// SIMATIC S7-200 project (STEP 7-Micro/WIN), CPU 221 REL 01.10

SYMBOL_TABLE USR1
Always_On        SM0.0    // This bit is always on.
Final_Count      VW0      // Variable memory word VW0 contains the ending value in the loop count (FINAL).
Initial_Count    VW10     // Variable memory word VW10 contains starting value in the loop count (INITIAL).
Current_Count    VW20     // Variable memory word VW20 contains the current loop count (INDEX).
First_Address    VB100    // Variable memory byte VB100 is the first address under which a value is saved.
END_SYMBOL_TABLE

ORGANIZATION_BLOCK MAIN:OB1
TITLE=
//  题目：设置位或字节的几种方法
// ***概述***
// 本程序描述了用一定值存入预定的存储区域或对预定的存储区域清零的几种方法
// 采用下列指令：
// *FILL           指令
// *FOR...NEXT     循环指令
// *RESET          指令
// 
// ***程序和注释***
// 本程序描述了用一定值存入预定的存储器位或字节，以及清除存储区内容的几种方法
// 采用下列指令：
// FILL          设置一个或几个字
// FOR...NEXT    FOR...NEXT循环
// R             对一位或几位置 0
// 
BEGIN
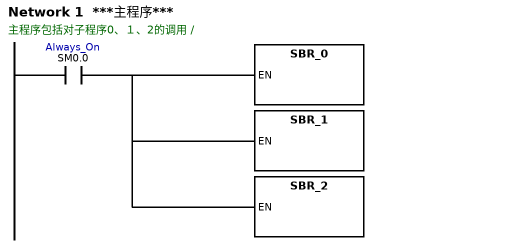
Network 1 // ***主程序***
// 主程序包括对子程序0、１、2的调用
// 
// SM0.0总是1
// 调用子程序0（FILL）
// 调用子程序1.（FOR...NEXT）
// 调用子程序2 （RESET）
LD     Always_On:SM0.0
CALL   SBR_0:SBR0
CALL   SBR_1:SBR1
CALL   SBR_2:SBR2
Network 2 // 主程序结束
// MEND				
// 
Network 3 // ***子程序0***
// 子程序0功能：如果输入I0.0=1,则把VW200中值复制到VW204至VW216
// 
Network 4 //  子程序1
// 当输入I0.1=1时，把几个初始数复制到变量存储区。
// 循环次数取决于VW10中的首次循环数和VW0中的最后一次循环数
// 当前循环次数存储在内存字VW20中
// 首次计数值（50）存储在累加器AC0中
// 计数值缓冲区首址（& VB100）存储在累加器AC1中，AC1为计数值缓冲区指针
// 每循环一次的功能：
// AC0的计数值存入AC1指针所指向的内存单元
// AC1指针加2个字节，指向下一个内存字
// AC0的计数值加4
// 直至最后一次循环
// 
Network 6 //  子程序2
// 如果输入I0.2=1,则把存储器位V100.0至V121.7及V204.0至V217.7置0
// 
END_ORGANIZATION_BLOCK

SUBROUTINE_BLOCK SBR_0:SBR0
TITLE=
BEGIN
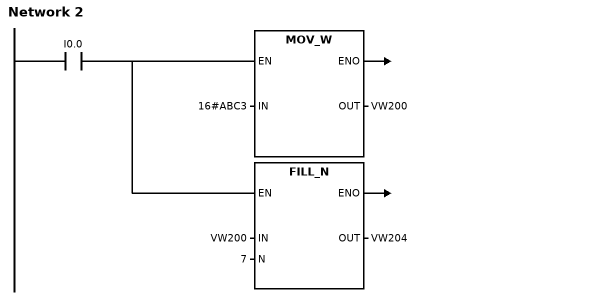
Network 2
// 读输入I0.0，如果I0.0=1,则
// 将十六进制数ABC3写入VW200
// 把VW200中值复制到VW204至VW216
LD     I0.0
MOVW   16#ABC3, VW200
FILL   VW200, VW204, 7
Network 3 //  子程序0结束
// RET					
// 
END_SUBROUTINE_BLOCK

SUBROUTINE_BLOCK SBR_1:SBR1
TITLE=
BEGIN
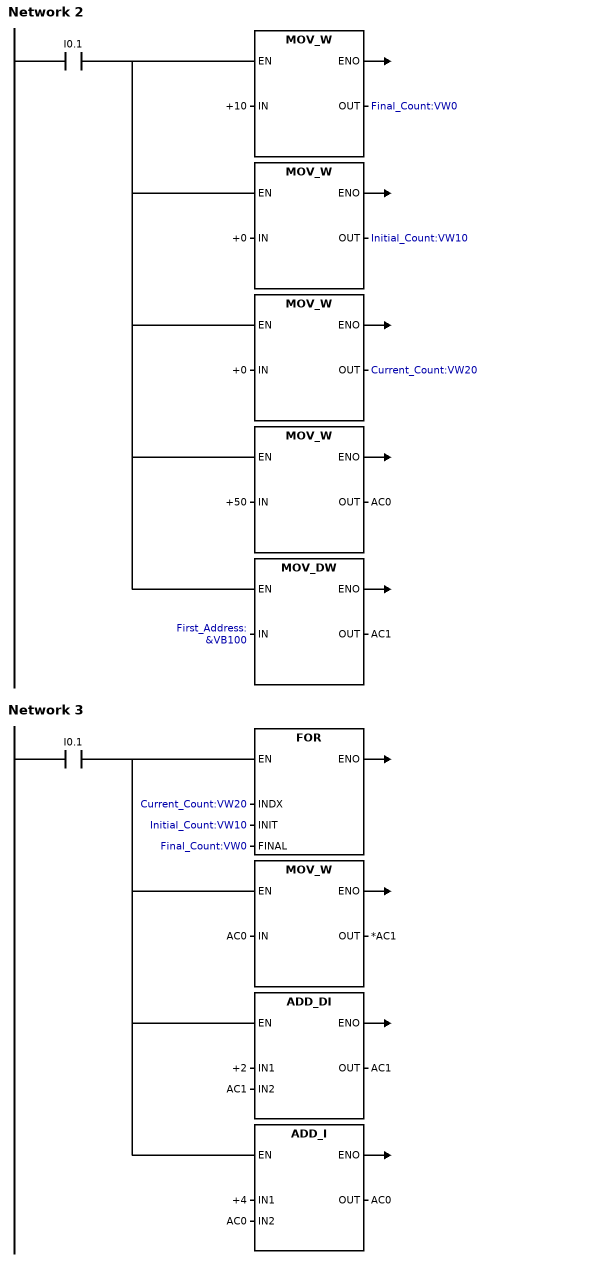
Network 2
// 读输入I0.1，如果I0.1=1,则
// 把最后一次循数环存入VW0
// 把第一次循环数存入VW10
// 把当前循环数存入VW20 (计数器)
// 首次计数值（50）存储在累加器0 (AC0)
// 累加器1（存储区指针）指向存储字节VW100
LD     I0.1
MOVW   +10, Final_Count:VW0
MOVW   +0, Initial_Count:VW10
MOVW   +0, Current_Count:VW20
MOVW   +50, AC0
MOVD   &First_Address:VB100, AC1
Network 3
// 循环开始
// 把当前计数值存到当前存储地址中
//AC1指针加2个字节，指向下一个内存字
//AC0的计数值加4
LD     I0.1
FOR    Current_Count:VW20, Initial_Count:VW10, Final_Count:VW0
MOVW   AC0, *AC1
+D     +2, AC1
+I     +4, AC0
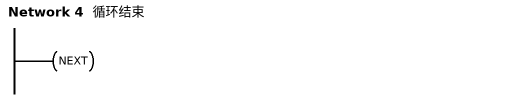
Network 4 // 循环结束
NEXT
Network 5 //  子程序1结束
// RET				
// 
END_SUBROUTINE_BLOCK

SUBROUTINE_BLOCK SBR_2:SBR2
TITLE=
BEGIN
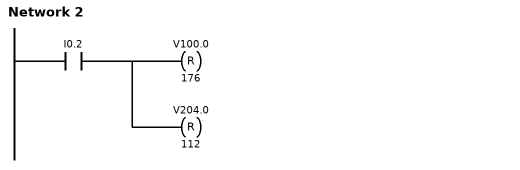
Network 2
// 读输入I0.2，如果I0.2=1,则 
// 把存储器位V100.0至V121.7置0
// V204.0至V217.7置0
LD     I0.2
R      V100.0, 176
R      V204.0, 112
Network 3 // 子程序2结束
// RET				
// 
END_SUBROUTINE_BLOCK
